(* CODESYS project exams.export

Project tree, tasks and I/O mapping:
  Device : CODESYS Control Win V3, 3S - Smart Software Solutions GmbH, version 3.5.16.30
    application Application
      libraries: Standard, * (System); CmpBitmapPool, * (System); VisuDialogs, * (System)
      task MainTask (cyclic, interval t#20ms, priority 2) calls PLC_PRG, watering, Capping, POU, door, door2, stopConveyerCondition, Labeling, GVLCAPINVISIBLE, Bank, BANKED_BOTTLE_XYPOSITION, stop_start, EmptySupply, terminal
      task VISU_TASK (cyclic, interval 100 ms, priority 31) calls VisuElems.Visu_Prg
      global variables GVL
      image pool ImagePool
      program Bank [FBD]
      program BANKED_BOTTLE_XYPOSITION [ST]
      program Capping [FBD]
      program door [ST]
      program door2 [FBD]
      program EmptySupply [FBD]
      program GVLCAPINVISIBLE [FBD]
      program Labeling [FBD]
      program PLC_PRG [SFC]: active_running, alarm_on, cappedBottleRunning, delaybeforeStart, fullBottleRunning, Initialize, labeledBottleRunning, restart
      program POU [ST]
      program stopConveyerCondition [FBD]
      program stop_start [FBD]
      program terminal [FBD]
      program watering [FBD]
      visualisation Visualization
  5ce3da45-db07-42e7-a21c-a00fff4ed8f6|370c3c75172605.Y3JvcCw4MDgsNjMyLDAsMA.bmp
  5ce3da45-db07-42e7-a21c-a00fff4ed8f6|370c3c75172605.Y3JvcCw4MDgsNjMyLDAsMA.jpg
  5ce3da45-db07-42e7-a21c-a00fff4ed8f6|cover14.jpg
  5ce3da45-db07-42e7-a21c-a00fff4ed8f6|empty.bmp
  5ce3da45-db07-42e7-a21c-a00fff4ed8f6|etiketa.bmp
  5ce3da45-db07-42e7-a21c-a00fff4ed8f6|etiketopoios.png
  5ce3da45-db07-42e7-a21c-a00fff4ed8f6|full.bmp
  5ce3da45-db07-42e7-a21c-a00fff4ed8f6|fullPacked.bmp
  5ce3da45-db07-42e7-a21c-a00fff4ed8f6|kapaki.bmp
  5ce3da45-db07-42e7-a21c-a00fff4ed8f6|labeled.bmp
  5ce3da45-db07-42e7-a21c-a00fff4ed8f6|logo.bmp
  5ce3da45-db07-42e7-a21c-a00fff4ed8f6|logo.jpg
  5ce3da45-db07-42e7-a21c-a00fff4ed8f6|logo1.bmp
  5ce3da45-db07-42e7-a21c-a00fff4ed8f6|stamped.bmp
  5ce3da45-db07-42e7-a21c-a00fff4ed8f6|tapotiras.bmp
  5ce3da45-db07-42e7-a21c-a00fff4ed8f6|Vikos-500x400.jpg
*)

// Device/Application/GVL
{attribute 'qualified_only'}
VAR_GLOBAL
	//photocell_2:BOOL;
	colorWater: DWORD;
	start:BOOL;//sima energopoiisis tainiodromou
	bottleInvisible:BOOL;
	bottlePosition :REAL;
	rotWheel:REAL;//peristrofi gia granazia
	waterMachineSwitch: BOOL; // diakoptis mixanis plirosis
	FullInvisible:BOOL;
	FullBottlePosition:REAL;
	capMachineSwitch:BOOL;// mixani kapakosis
	capMove:INT;
	rotDoor:INT; // peristrofi portas
	doorSwitch:BOOL;//diakoptis trofodosias me adeies fiales
	openDoor:BOOL;//
	closeDoor:BOOL;
	stopforCapping:BOOL;
	stopforWatering:BOOL;
	CapInvisible: BOOL;
	CapBottlePosition:REAL;
	labelMove:INT;
	labelingMachineSwitch:BOOL;// diakoptis mixanis etiketas
	stopforLabeling:BOOL;
	LabelInvisible: BOOL;
	Inserted_Bottles_Counter:WORD;
	XlabelBottlePosition:REAL;
	YlabelBottlePosition:REAL;
	Stop:BOOL;// sima ektaktis diakopis
	BANKFULL:BOOL;// i trapeza gemise
	BANKCAPACITY:INT;//xoritikotita trapezas
	BANKEDBOTTLES:WORD;// posa mpoukalia etoimastikan
	BankSwitcher:BOOL;// diakoptis trapezas apothesis
	restartConveyerSignal:BOOL;// sima epanenergopoiisis tainiodromou
	userInputBottles:INT; // arithmos mpoukaliwn pou tha gemisei o xeiristis
	BottleArsenal:INT;// arithmos mpoukaliwn trofodosias
	ALARM:BOOL; // sirina aneparkeis trofodosia me mpoykalia
	START_STOP:BOOL; // start and not(stop)
	ALARMFULLBANK:BOOL;//sinagermos gemati trapeza
	del:BOOL; // zestama ekinnisis
	terminalCondition:BOOL;// termatiki sinthiki diakopis
	interruption:BOOL; //diakopi logo gematis trapezas
	
END_VAR

// Device/Application/PLC_PRG
PROGRAM PLC_PRG
VAR

	
	delaybefore: TON;
END_VAR

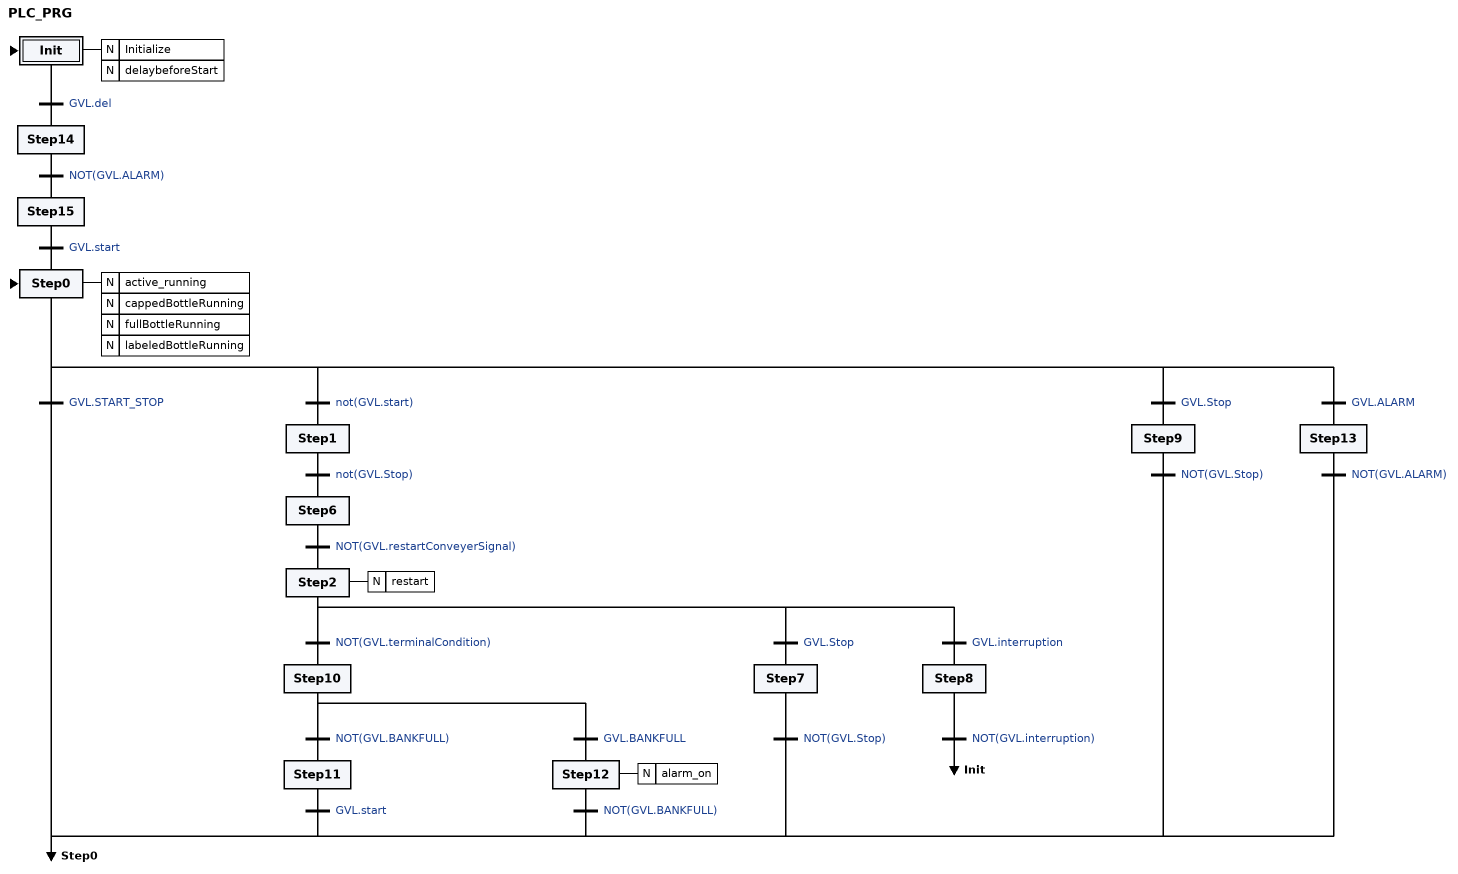
INITIAL_STEP Init:
    Initialize(N);
    delaybeforeStart(N);
END_STEP
TRANSITION FROM Init TO Step14
    := GVL.del;
END_TRANSITION
STEP Step14:
END_STEP
TRANSITION FROM Step14 TO Step15
    := NOT(GVL.ALARM);
END_TRANSITION
STEP Step15:
END_STEP
TRANSITION FROM Step15 TO Step0
    := GVL.start;
END_TRANSITION
STEP Step0:
    active_running(N);
    cappedBottleRunning(N);
    fullBottleRunning(N);
    labeledBottleRunning(N);
END_STEP
TRANSITION FROM Step0 TO Step0
    := GVL.START_STOP;
END_TRANSITION
TRANSITION FROM Step0 TO Step1
    := not(GVL.start);
END_TRANSITION
STEP Step1:
END_STEP
TRANSITION FROM Step1 TO Step6
    := not(GVL.Stop);
END_TRANSITION
STEP Step6:
END_STEP
TRANSITION FROM Step6 TO Step2
    := NOT(GVL.restartConveyerSignal);
END_TRANSITION
STEP Step2:
    restart(N);
END_STEP
TRANSITION FROM Step2 TO Step10
    := NOT(GVL.terminalCondition);
END_TRANSITION
STEP Step10:
END_STEP
TRANSITION FROM Step10 TO Step11
    := NOT(GVL.BANKFULL);
END_TRANSITION
STEP Step11:
END_STEP
TRANSITION FROM Step11 TO Step0
    := GVL.start;
END_TRANSITION
TRANSITION FROM Step10 TO Step12
    := GVL.BANKFULL;
END_TRANSITION
STEP Step12:
    alarm_on(N);
END_STEP
TRANSITION FROM Step12 TO Step0
    := NOT(GVL.BANKFULL);
END_TRANSITION
TRANSITION FROM Step2 TO Step7
    := GVL.Stop;
END_TRANSITION
STEP Step7:
END_STEP
TRANSITION FROM Step7 TO Step0
    := NOT(GVL.Stop);
END_TRANSITION
TRANSITION FROM Step2 TO Step8
    := GVL.interruption;
END_TRANSITION
STEP Step8:
END_STEP
TRANSITION FROM Step8 TO Init
    := NOT(GVL.interruption);
END_TRANSITION
TRANSITION FROM Step0 TO Step9
    := GVL.Stop;
END_TRANSITION
STEP Step9:
END_STEP
TRANSITION FROM Step9 TO Step0
    := NOT(GVL.Stop);
END_TRANSITION
TRANSITION FROM Step0 TO Step13
    := GVL.ALARM;
END_TRANSITION
STEP Step13:
END_STEP
TRANSITION FROM Step13 TO Step0
    := NOT(GVL.ALARM);
END_TRANSITION

ACTION active_running:
IF( (GVL.userInputBottles>=(GVL.BANKEDBOTTLES+3))AND(NOT(GVL.BANKFULL))) THEN //EDW BANKFULL
GVL.bottlePosition := GVL.bottlePosition +0.2;
END_IF
IF( GVL.START_STOP) THEN
GVL.rotWheel:=GVL.rotWheel+10;
END_IF
//IF (watering.InsertedBottles.CV>1)THEN 
	//GVL.FullBottlePosition:=GVL.FullBottlePosition+0.2;
//END_IF

//IF (watering.InsertedBottles.CV >2) THEN
	//GVL.CapBottlePosition:=GVL.CapBottlePosition+0.2;
//END_IF
END_ACTION

ACTION alarm_on:
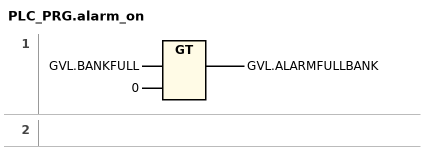
// NETWORK 1
GVL.ALARMFULLBANK := GVL.BANKFULL > 0;

// NETWORK 2
END_ACTION

ACTION cappedBottleRunning:
IF ((watering.InsertedBottles.CV >=2)AND(GVL.userInputBottles>=(GVL.BANKEDBOTTLES+1))AND(NOT(GVL.BANKFULL))) THEN
	GVL.CapBottlePosition:=GVL.CapBottlePosition+0.2;
END_IF
END_ACTION

ACTION delaybeforeStart:
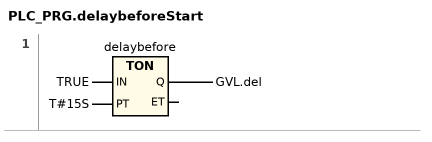
// NETWORK 1
delaybefore(IN := TRUE, PT := T#15S); // TON
GVL.del := delaybefore.Q;
END_ACTION

ACTION fullBottleRunning:
IF ((watering.InsertedBottles.CV>=1)AND(GVL.userInputBottles>=(2+GVL.BANKEDBOTTLES))AND(NOT(GVL.BANKFULL)))THEN //EDW BANKFULL
	GVL.FullBottlePosition:=GVL.FullBottlePosition+0.2;
END_IF
END_ACTION

ACTION Initialize:
GVL.colorWater :=16#FFB0E0E6;
GVL.FullInvisible:=TRUE;
GVL.bottleInvisible:=TRUE;
GVL.capMachineSwitch:=FALSE;
GVL.CapInvisible:=TRUE;
GVL.LabelInvisible:=TRUE;
GVL.waterMachineSwitch:=FALSE;
GVL.labelingMachineSwitch :=FALSE;
GVL.BankSwitcher:=FALSE;
GVL.BottleArsenal:=200;
GVL.BANKCAPACITY:=110;
END_ACTION

ACTION labeledBottleRunning:
IF ((watering.InsertedBottles.CV >=3) AND(GVL.userInputBottles>GVL.BANKEDBOTTLES)) THEN
	GVL.XlabelBottlePosition:=GVL.XlabelBottlePosition+0.2;
END_IF
END_ACTION

ACTION restart:
GVL.bottlePosition:=0;
GVL.start:=TRUE;
//GVL.FullInvisible:=FALSE;
GVL.FullBottlePosition:=0;
GVL.capMove:=0;
GVL.CapBottlePosition:=0;
//IF (watering.InsertedBottles.CV >1) THEN
	//GVL.CapInvisible:=FALSE;
//END_IF

GVL.labelMove:=0;
//IF (watering.InsertedBottles.CV >2) THEN
//GVL.LabelInvisible:=FALSE;		
//END_IF
GVL.XlabelBottlePosition:=0;
GVL.YlabelBottlePosition:=0;
END_ACTION

END_PROGRAM

// Device/Application/watering
PROGRAM watering
VAR
	WaterProcess: TON;
	fill: RS;
	InsertedBottles:CTU;
END_VAR
VAR // added by the converter: edge detectors and wires of the graphical bodies
    _w1 : BOOL;
END_VAR

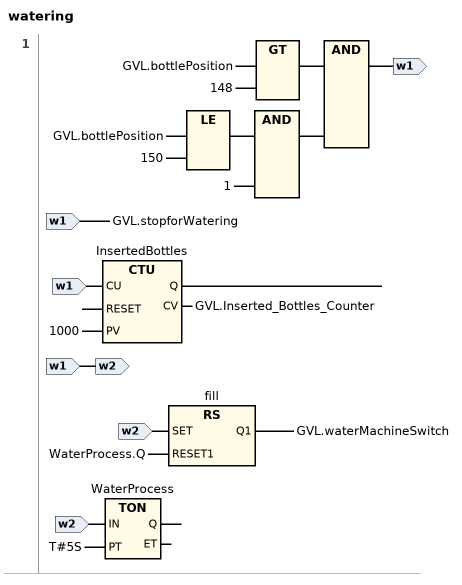
// NETWORK 1
_w1 := GVL.bottlePosition > 148 AND (GVL.bottlePosition <= 150 AND 1);
GVL.stopforWatering := _w1;
InsertedBottles(CU := _w1, PV := 1000, CV => GVL.Inserted_Bottles_Counter); // CTU
fill(SET := _w1, RESET1 := WaterProcess.Q); // RS
GVL.waterMachineSwitch := fill.Q1;
WaterProcess(IN := _w1, PT := T#5S); // TON

END_PROGRAM

// Device/Application/Capping
PROGRAM Capping
VAR_INPUT
	
	CapProcess: TON;
	cap: RS;
END_VAR

VAR
	NumberOfCaps: CTU;
END_VAR
VAR // added by the converter: edge detectors and wires of the graphical bodies
    _w1 : BOOL;
END_VAR

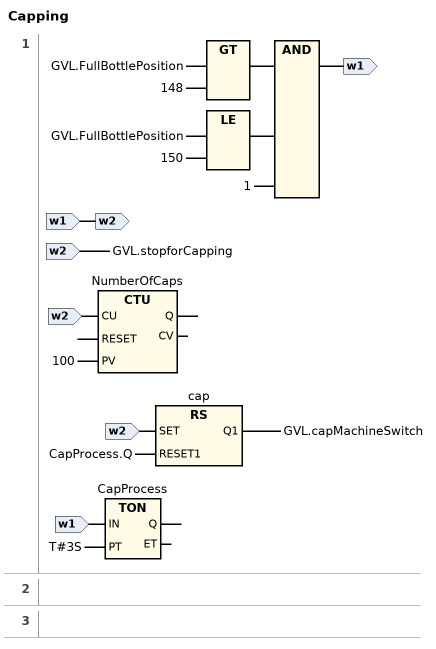
// NETWORK 1
_w1 := GVL.FullBottlePosition > 148 AND GVL.FullBottlePosition <= 150 AND 1;
GVL.stopforCapping := _w1;
NumberOfCaps(CU := _w1, PV := 100); // CTU
cap(SET := _w1, RESET1 := CapProcess.Q); // RS
GVL.capMachineSwitch := cap.Q1;
CapProcess(IN := _w1, PT := T#3S); // TON

// NETWORK 2

// NETWORK 3

END_PROGRAM

// Device/Application/POU
PROGRAM POU
VAR
END_VAR

IF ( GVL.capMachineSwitch =TRUE) THEN
	GVL.capMove:=40;
	//GVL.labelMove:=40;
	END_IF
IF(GVL.labelingMachineSwitch=TRUE)THEN
	GVL.labelMove:=40;
END_IF
IF (Capping.cap.RESET1) THEN
	GVL.capMove:=0;
END_IF
IF (Labeling.label.RESET1) THEN
	GVL.labelMove:=0;
END_IF

END_PROGRAM

// Device/Application/Labeling
PROGRAM Labeling
VAR
	LabelProcess: TON;
	label: RS;
	NumberOfLabels: CTU;
END_VAR
VAR // added by the converter: edge detectors and wires of the graphical bodies
    _w1 : BOOL;
END_VAR

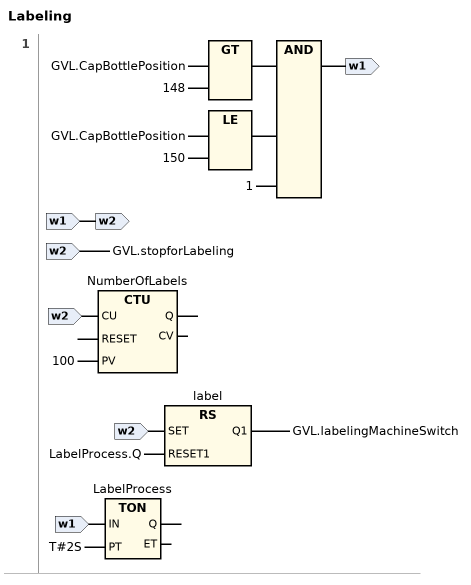
// NETWORK 1
_w1 := GVL.CapBottlePosition > 148 AND GVL.CapBottlePosition <= 150 AND 1;
GVL.stopforLabeling := _w1;
NumberOfLabels(CU := _w1, PV := 100); // CTU
label(SET := _w1, RESET1 := LabelProcess.Q); // RS
GVL.labelingMachineSwitch := label.Q1;
LabelProcess(IN := _w1, PT := T#2S); // TON

END_PROGRAM

// Device/Application/door
PROGRAM door
VAR
	DELAY:TON;
END_VAR

IF( GVL.openDoor) THEN
	GVL.rotDoor:=-90;
	IF(GVL.closeDoor) THEN
		GVL.rotDoor:=0;
	END_IF
END_IF

END_PROGRAM

// Device/Application/door2
PROGRAM door2
VAR
	porta: TON;
END_VAR
VAR // added by the converter: edge detectors and wires of the graphical bodies
    _w1 : BOOL;
END_VAR

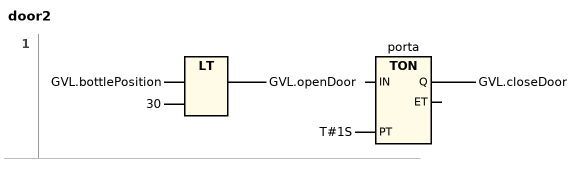
// NETWORK 1
_w1 := GVL.bottlePosition < 30;
GVL.openDoor := _w1;
porta(IN := _w1, PT := T#1S); // TON
GVL.closeDoor := porta.Q;

END_PROGRAM

// Device/Application/stopConveyerCondition
PROGRAM stopConveyerCondition
VAR
	Standard_Stop: RS;
	Standard_Delay: TON;
END_VAR
VAR // added by the converter: edge detectors and wires of the graphical bodies
    _w1 : BOOL;
END_VAR

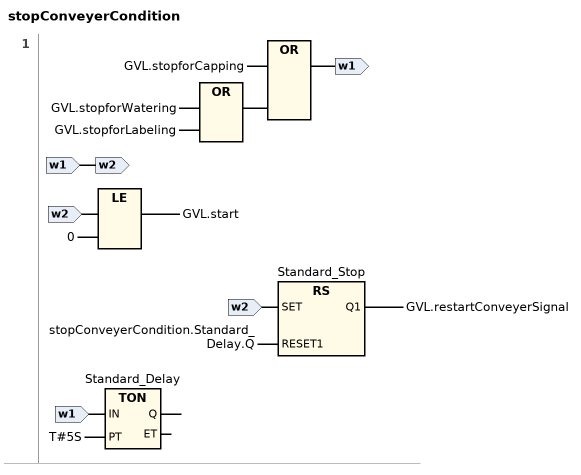
// NETWORK 1
_w1 := GVL.stopforCapping OR (GVL.stopforWatering OR GVL.stopforLabeling);
GVL.start := _w1 <= 0;
Standard_Stop(SET := _w1, RESET1 := stopConveyerCondition.Standard_Delay.Q); // RS
GVL.restartConveyerSignal := Standard_Stop.Q1;
Standard_Delay(IN := _w1, PT := T#5S); // TON

END_PROGRAM

// Device/Application/GVLCAPINVISIBLE
PROGRAM GVLCAPINVISIBLE
VAR
END_VAR

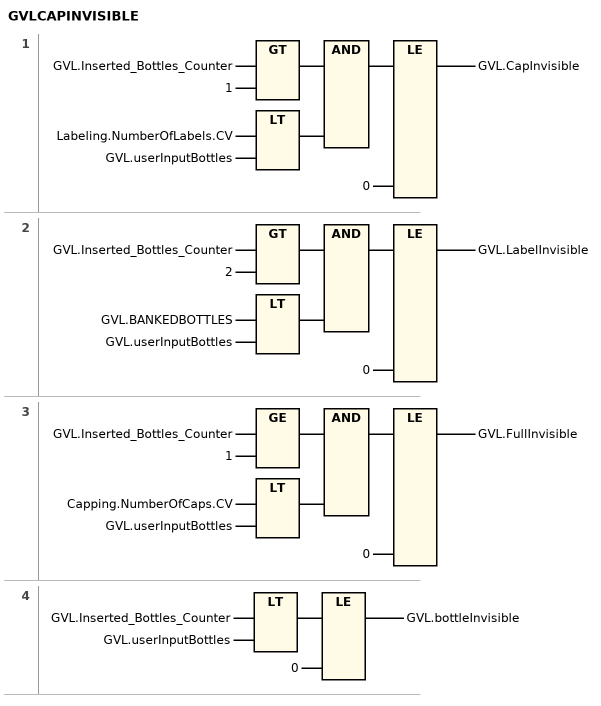
// NETWORK 1
GVL.CapInvisible := (GVL.Inserted_Bottles_Counter > 1 AND Labeling.NumberOfLabels.CV < GVL.userInputBottles) <= 0;

// NETWORK 2
GVL.LabelInvisible := (GVL.Inserted_Bottles_Counter > 2 AND GVL.BANKEDBOTTLES < GVL.userInputBottles) <= 0;

// NETWORK 3
GVL.FullInvisible := (GVL.Inserted_Bottles_Counter >= 1 AND Capping.NumberOfCaps.CV < GVL.userInputBottles) <= 0;

// NETWORK 4
GVL.bottleInvisible := (GVL.Inserted_Bottles_Counter < GVL.userInputBottles) <= 0;

END_PROGRAM

// Device/Application/Bank
PROGRAM Bank
VAR
	BANKCONTROLLER: CTU;
	BANKSWITCH: RS;
	BANKDELAY: TON;
END_VAR
VAR // added by the converter: edge detectors and wires of the graphical bodies
    _w1 : BOOL;
END_VAR

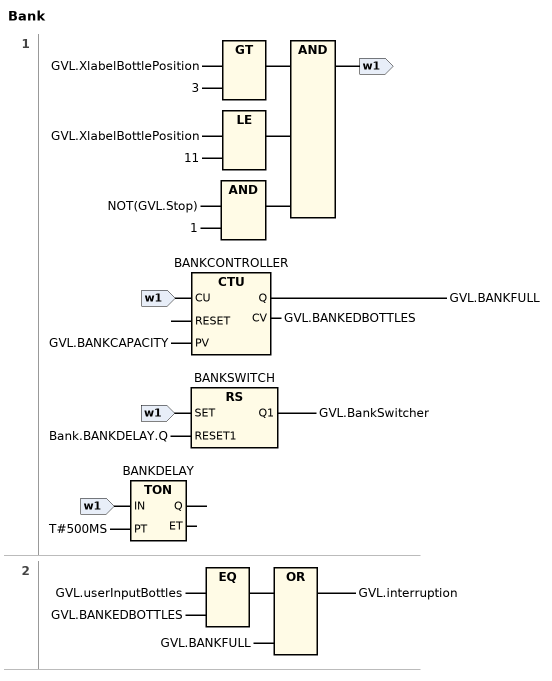
// NETWORK 1
_w1 := GVL.XlabelBottlePosition > 3 AND GVL.XlabelBottlePosition <= 11 AND ((NOT(GVL.Stop)) AND 1);
BANKCONTROLLER(CU := _w1, PV := GVL.BANKCAPACITY, CV => GVL.BANKEDBOTTLES); // CTU
GVL.BANKFULL := BANKCONTROLLER.Q;
BANKSWITCH(SET := _w1, RESET1 := Bank.BANKDELAY.Q); // RS
GVL.BankSwitcher := BANKSWITCH.Q1;
BANKDELAY(IN := _w1, PT := T#500MS); // TON

// NETWORK 2
GVL.interruption := GVL.userInputBottles = GVL.BANKEDBOTTLES OR GVL.BANKFULL;

END_PROGRAM

// Device/Application/BANKED_BOTTLE_XYPOSITION
PROGRAM BANKED_BOTTLE_XYPOSITION
VAR
END_VAR

IF(Bank.BANKSWITCH.SET) THEN
	GVL.YlabelBottlePosition:=90;
END_IF

END_PROGRAM

// Device/Application/stop_start
PROGRAM stop_start
VAR
END_VAR

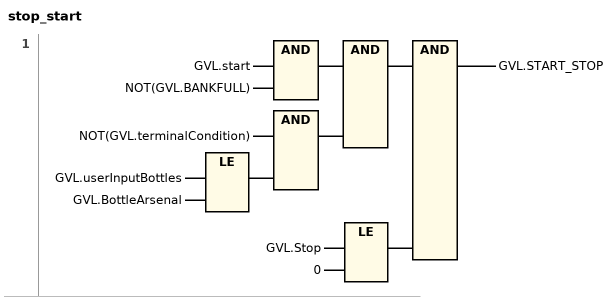
// NETWORK 1
GVL.START_STOP := ((GVL.start AND (NOT(GVL.BANKFULL))) AND ((NOT(GVL.terminalCondition)) AND GVL.userInputBottles <= GVL.BottleArsenal)) AND GVL.Stop <= 0;

END_PROGRAM

// Device/Application/EmptySupply
PROGRAM EmptySupply
VAR
END_VAR

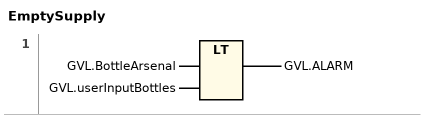
// NETWORK 1
GVL.ALARM := GVL.BottleArsenal < GVL.userInputBottles;

END_PROGRAM

// Device/Application/terminal
PROGRAM terminal
VAR
END_VAR

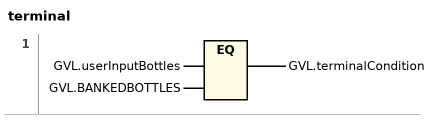
// NETWORK 1
GVL.terminalCondition := GVL.userInputBottles = GVL.BANKEDBOTTLES;

END_PROGRAM

// Device/Application/Visualization
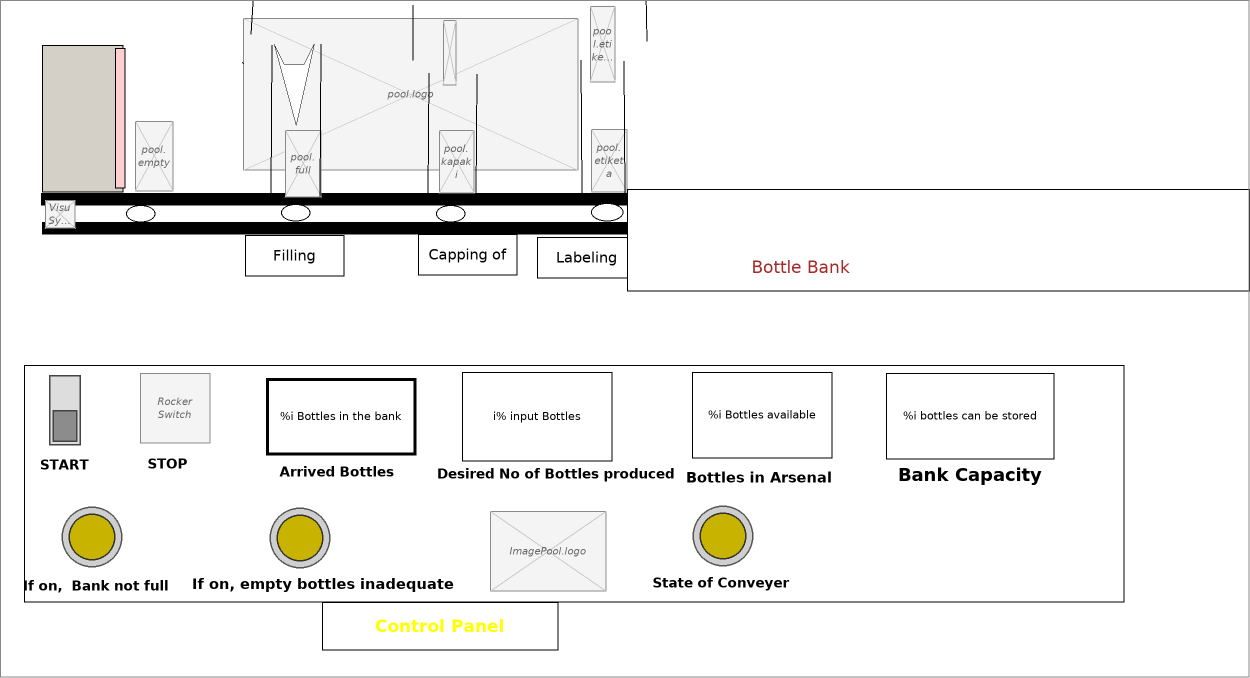
VISUALIZATION Visualization  // 1250x678
    Rectangle (41,193 650x12)
    Rectangle (42,222 650x12)
    Image (662,199 25x29), image: VisuSymbols.Symbols.Wheel
        p2858320360: GVL.rotWheel
    Image (45,200 30x28), image: VisuSymbols.Symbols.Wheel
        p2858320360: GVL.rotWheel
    Rectangle (687,193 13x41)
    Image (243,18 335x152), image: pool.logo
    Ellipse (126,205 29x17)
    Ellipse (281,204 29x17)
    Ellipse (591,203 32x18)
    Ellipse (436,205 29x17)
    RoundedRectangle (42,45 81x147)
    Rectangle (115,48 10x140)
        p2858320360: GVL.rotDoor
    Image (135,121 38x70), invisible if: GVL.bottleInvisible, image: pool.empty
        p3560616238: GVL.bottlePosition
    Image (285,130 36x67), invisible if: GVL.FullInvisible, image: pool.full
        p3560616238: GVL.FullBottlePosition
    Image (439,130 35x63), invisible if: GVL.CapInvisible, image: pool.kapaki
        p3560616238: GVL.CapBottlePosition
    Image (591,129 36x63), invisible if: GVL.LabelInvisible, image: pool.etiketa
        p3560616238: GVL.XlabelBottlePosition
        p2738717112: GVL.YlabelBottlePosition
    Rectangle (245,235 99x41), "Filling"
    Rectangle (418,234 99x41), "Capping of"
    Rectangle (537,237 99x41), "Labeling"
    Polyline (242,62) (243,63)
    Line (269,45)
    Line (271,194) (272,45)
    Line (320,196) (321,44)
    Line (251,34) (255,-28)
    Polygon (274,44) (296,125) (314,44) (304,64) (284,64), colour toggle: GVL.waterMachineSwitch
        p2167032090: GVL.colorWater
    Line (428,195) (429,73)
    Line (476,196) (477,74)
    Line (413,60) (413,5)
    Image (443,20 13x65), image: pool.tapotiras
        p2738717112: GVL.capMove
    Line (582,193) (581,60)
    Line (625,196) (624,61)
    Image (590,6 25x76), image: pool.etiketopoios
        p2738717112: GVL.labelMove
    Line (647,41) (646,-7)
    RoundedRectangle (627,189 623x102)
    Label (726,252 150x30), "Bottle Bank"
    Rectangle (24,365 1100x237)
    Label (37,450 55x30), "START"
    Label (140,449 55x30), "STOP"
    RockerSwitch (140,373 70x70), variable: GVL.Stop, behaviour: TOGGLE, style: Switch-RockerSwitch-Gray
    DipSwitch (30,375 70x70), variable: GVL.start, behaviour: TOGGLE, style: Switch-DipSwitch-Gray
    Rectangle (266,378 150x77), "%i Bottles in the bank", text variable: GVL.BANKEDBOTTLES
    Rectangle (462,372 150x89), "i% input Bottles", text variable: GVL.userInputBottles
        OnMouseClick: write the text variable via Default
    Lamp1 (688,501 70x70), variable: GVL.START_STOP, style: Lamp-Lamp1-Yellow
    Label (262,457 150x30), "Arrived Bottles"
    Label (442,459 228x30), "Desired No of Bottles produced"
    Lamp1 (57,502 70x70), variable: NOT(GVL.BANKFULL), style: Lamp-Lamp1-Yellow
    Label (21,571 150x30), "If on, Bank not full"
    Lamp1 (265,503 70x70), variable: GVL.ALARM, style: Lamp-Lamp1-Yellow
    Label (179,569 288x30), "If on, empty bottles inadequate"
    Label (646,568 150x30), "State of Conveyer"
    Image (490,511 116x80), image: ImagePool.logo
    Rectangle (322,602 236x48), "Control Panel"
    RoundedRectangle (692,372 140x86), "%i Bottles available", text variable: GVL.BottleArsenal
    Label (682,464 154x27), "Bottles in Arsenal"
    RoundedRectangle (886,373 168x86), "%i bottles can be stored", text variable: GVL.BANKCAPACITY
    Label (895,459 150x32), "Bank Capacity"
END_VISUALIZATION
